{attribute 'linkalways'} 
{attribute 'no_explicit_call' := 'This FB is a CLASS and must be accessed using methods or properties'}
{attribute 'enable_dynamic_creation'}
FUNCTION_BLOCK Node_F_VN_RegionOrientation EXTENDS VisionNode
VAR
    ipSrcImage : _ITcVnImage;
    stOrientation : _TcVnRotatedRectangle;
    hrPrev : _HRESULT(S_OK);
	hresult : _HRESULT(S_OK);
END_VAR

METHOD PUBLIC  Clone : I_Node
VAR
	pNode : POINTER TO Node_F_VN_RegionOrientation;
END_VAR
pNode := __NEW(Node_F_VN_RegionOrientation);
Clone := pNode^;
END_METHOD

METHOD FB_init : BOOL
VAR_INPUT
	bInitRetains : BOOL; // if TRUE, the retain variables are initialized (warm start / cold start)
	bInCopyCode : BOOL;  // if TRUE, the instance afterwards gets moved into the copy code (online change)
END_VAR
AddInput('ipSrcImage', ipSrcImage);
AddInput('hrPrev', hrPrev);
AddOutput('stOrientation', stOrientation);
AddOutput('hresult', hresult);
END_METHOD

METHOD PROTECTED OnExecute
hresult.Value := F_VN_RegionOrientation(
	ipSrcImage := ipSrcImage.Value,
    stOrientation := stOrientation.Value,
	hrPrev:= hrPrev.Value);
END_METHOD

METHOD PUBLIC PreExecutionCheck
VAR_INPUT
	Check : I_PreExecutionChecks;
END_VAR
Check.IsTrue(ipSrcImage.IsValid, 'ipSrcImage must contain an image');
Check.IsTrue(ipSrcImage.HasChannelCount(1), 'ipSrcImage must contain 1 channel');
END_METHOD

END_FUNCTION_BLOCK

(* stored: Version 1.1.0.1, ProductVersion 3.1.4024.13
   POU Node_F_VN_RegionOrientation: Id {60984004-c404-0d29-0701-0fccf367044f}, SpecialFunc None
   Folder Constructor: Id {1344e5e3-37bf-0692-0e3c-97bb78a25be1}
   Method Clone: Id {02e02bcc-33b5-052e-2b7c-7e017337cfc4}
   Method FB_init: Id {2dc8054e-6cbc-0d05-16f8-0727a1a8b5d4}
   Method OnExecute: Id {03ad62fa-bdb8-0e59-202d-e11ff414347c}
   Method PreExecutionCheck: Id {0e2a84e5-9dbc-07cb-01fd-894060664cd8} *)
